TYPE Terminal_Group_Input_typ : 	
	STRUCT 
		Par : Terminal_Group_Parameter_typ;
	END_STRUCT
END_TYPE

(* stored: Version 1.1.0.1, ProductVersion 3.1.4024.3
   DUT Terminal_Group_Input_typ: Id {f5a0ad06-13f4-0839-0024-729e63b144ad} *)
